FUNCTION_BLOCK FB_Bender
VAR_IN_OUT
    stBender : ST_MotionStage;
    bSTOEnable1 : BOOL;
    bSTOEnable2 : BOOL;
END_VAR
VAR_INPUT
END_VAR
VAR_OUTPUT
END_VAR
VAR
END_VAR

// Simple FB to tie stBender.bHardwareEnable to STO
// Originally part of FB_RunHOMS, but want to use this for all systems, not all of which have a bender motor
stBender.bHardwareEnable := bSTOEnable1 AND bSTOEnable2;

END_FUNCTION_BLOCK

(* stored: Version 1.1.0.1, ProductVersion 3.1.4024.12
   POU FB_Bender: Id {d1d24e90-e8bb-4e37-9db9-9aec40d6deb9}, SpecialFunc None *)
